// TIA Portal V17 export
// export: Created 2022-07-20T07:02:31.4890995Z, ExportSetting WithDefaults, DisplayName Totally Integrated Automation Portal, DisplayVersion V17, DisplayName TIA Portal Openness, DisplayVersion V17, DisplayName TIA Portal Version Control Interface, DisplayVersion V17, DisplayName SINAMICS Startdrive Advanced, DisplayVersion V17, DisplayName SINAMICS Startdrive G130, G150, S120, S150, SINAMICS MV, S210, DisplayVersion V17, DisplayName SINAMICS Startdrive G110M, G120, G120C, G120D, G120P, G115D, DisplayVersion V17, DisplayName STEP 7 Professional, DisplayVersion V17, DisplayName STEP 7 Safety, DisplayVersion V17, DisplayName WinCC Advanced, DisplayVersion V17
FUNCTION_BLOCK "FB11004_ProfileDataFifo"   // FB11004, LAD
TITLE = FIFO
{ S7_Optimized_Access := 'TRUE' }
VERSION : 0.1
// stored: AutoNumber false, IsIECCheckEnabled false, IsRetainMemResEnabled false, MemoryReserve 100, SetENOAutomatically false, UDAEnableTagReadback false
   VAR_INPUT
      GetProfile { ExternalAccessible := 'False'; ExternalVisible := 'False'; ExternalWritable := 'False'} : Bool;
      State { ExternalAccessible := 'False'; ExternalVisible := 'False'; ExternalWritable := 'False'} : UInt;
      Profile { ExternalAccessible := 'False'; ExternalVisible := 'False'; ExternalWritable := 'False'} : "stSheetProfile";
   END_VAR
   VAR_OUTPUT
      ItemsNumber { ExternalAccessible := 'False'; ExternalVisible := 'False'; ExternalWritable := 'False'} : UInt;
      ProfileAvailable { ExternalAccessible := 'False'; ExternalVisible := 'False'; ExternalWritable := 'False'} : Bool;
      Status { ExternalAccessible := 'False'; ExternalVisible := 'False'; ExternalWritable := 'False'} : UInt;
      ActualProfile { ExternalAccessible := 'False'; ExternalVisible := 'False'; ExternalWritable := 'False'} : "stSheetProfile";
   END_VAR
   VAR
      statFifo : Array[1.."MAX_IFOIL_FIFO_ITEMS_NUMBER"] of "stSheetProfile";
      statItemNumber { S7_SetPoint := 'True'} : UInt := 0;
      R_TRIG_GetProfile : R_TRIG;
      R_TRIG_GetDataFifo { S7_SetPoint := 'True'} : R_TRIG;
      statLastItem { S7_SetPoint := 'True'} : Bool;
   END_VAR
   VAR_TEMP
      FifoNumber : UInt;   // NextProfileTo
      AreaNumber : UInt;
   END_VAR
BEGIN

REGION Network 1 (SCL): Comments
   //==========================================================================================
   // SIEMENS SAS      RC-FR DI FA APC
   //------------------------------------------------------------------------------------------
   // Restrictions:    TIA V16 and more
   // Requirements:    S7-1500 - MGI Library
   // Functionality:   This function block offers fifo functionnality for stSheetProfile
   //------------------------------------------------------------------------------------------
   // Change log table:
   // Version      Date        Expert in charge    Changes applied
   // 01.00.01     09.06.2020  RTO                 First released version
   //==========================================================================================
END_REGION

REGION Network 2 (SCL): First Scan
   IF "FirstScan" THEN

       // Clear Interface
       #Status := 16#0;
       #ItemsNumber := "MAX_IFOIL_FIFO_ITEMS_NUMBER";
       #ProfileAvailable := FALSE;

       #ActualProfile.Length := 0.0;
       #ActualProfile.StampAreaStartAdjustment := 0.0;
       FOR #AreaNumber := 1 TO "MAX_NUMBER_OF_FOIL_AREA" DO
           #ActualProfile.Area[#AreaNumber].Start := 0.0;
           #ActualProfile.Area[#AreaNumber].End := 0.0;
       END_FOR;

       // Clear Fifo
       FOR #FifoNumber := 1 TO "MAX_IFOIL_FIFO_ITEMS_NUMBER" DO
           #statFifo[#FifoNumber].Length := 0.0;
           #statFifo[#FifoNumber].StampAreaStartAdjustment := 0.0;
           FOR #AreaNumber := 1 TO "MAX_NUMBER_OF_FOIL_AREA" DO
               #statFifo[#FifoNumber].Area[#AreaNumber].Start := 0.0;
               #statFifo[#FifoNumber].Area[#AreaNumber].End := 0.0;
           END_FOR;
       END_FOR;

       #statItemNumber := 0;
       #statLastItem := FALSE;

   END_IF;
END_REGION

REGION Network 3 (SCL): Edge Signal Management
   REGION EDGE SIGNALS
       #R_TRIG_GetProfile(CLK := #GetProfile);
       #R_TRIG_GetDataFifo(CLK := #State = 1 AND #statItemNumber < "MAX_IFOIL_FIFO_ITEMS_NUMBER" AND NOT #R_TRIG_GetProfile.Q);
   END_REGION
END_REGION

REGION Network 4 (SCL): Manage Fifo ready
   IF #State = 0 AND (#Status = 1 OR #Status = 2)
   THEN
       #Status := 0;
   END_IF;
END_REGION

REGION Network 5 (SCL): Put data in Fifo
   IF #State = 1 AND #statItemNumber < "MAX_IFOIL_FIFO_ITEMS_NUMBER" AND NOT #R_TRIG_GetProfile.Q THEN

       IF #R_TRIG_GetDataFifo.Q THEN
           // Get profile
           #statFifo[#statItemNumber + 1] := #Profile;

           // increase number of items
           #statItemNumber := #statItemNumber + 1;

       END_IF;

       // Send status
       #Status := 1;
   END_IF;
END_REGION

REGION Network 6 (SCL): Clear Fifo data
   IF #State = 2 AND #statItemNumber > 0 AND NOT #R_TRIG_GetProfile.Q THEN

       // Clear Fifo
       FOR #FifoNumber := 1 TO "MAX_IFOIL_FIFO_ITEMS_NUMBER" DO
           #statFifo[#FifoNumber].Length := 0.0;
           #statFifo[#FifoNumber].StampAreaStartAdjustment := 0.0;
           FOR #AreaNumber := 1 TO "MAX_NUMBER_OF_FOIL_AREA" DO
               #statFifo[#FifoNumber].Area[#AreaNumber].Start := 0.0;
               #statFifo[#FifoNumber].Area[#AreaNumber].End := 0.0;
           END_FOR;
       END_FOR;

       // Reset number of items
       #statItemNumber := 0;

       // Send status
       #Status := 2;

   END_IF;
END_REGION

REGION Network 7 (SCL): Get data from Fifo
   IF #R_TRIG_GetProfile.Q THEN

       // Get profile in Fifo
       #ActualProfile := #statFifo[1];

       IF #statItemNumber >= 2 THEN
           // Go up values in Fifo
           FOR #FifoNumber := 2 TO #statItemNumber DO
               #statFifo[#FifoNumber - 1] := #statFifo[#FifoNumber];
           END_FOR;
       END_IF;

       // Check if last item
       #statLastItem := #statItemNumber = 1;

       IF #statItemNumber >= 1 THEN
           // Clear last profile
           #statFifo[#statItemNumber].Length := 0.0;
           #statFifo[#statItemNumber].StampAreaStartAdjustment := 0.0;
           FOR #AreaNumber := 1 TO "MAX_NUMBER_OF_FOIL_AREA" DO
               #statFifo[#statItemNumber].Area[#AreaNumber].Start := 0.0;
               #statFifo[#statItemNumber].Area[#AreaNumber].End := 0.0;
           END_FOR;

           // Decrease number of items
           #statItemNumber := #statItemNumber - 1;
       END_IF;

   END_IF;
END_REGION

REGION Network 8: Manage profile available information
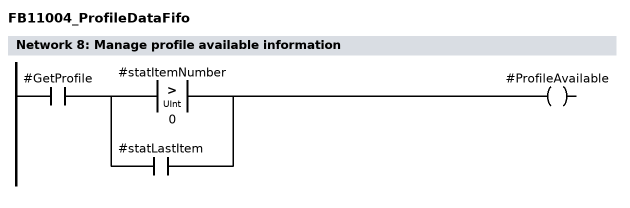
   RUNG wire#powerrail
      Contact( #GetProfile )
      wire#w1
      { S7_Templates := "SrcType := UInt" } GT_Contact(in1 := #statItemNumber, in2 := 0)
      wire#w2
      Coil( #ProfileAvailable )
   END_RUNG
   RUNG wire#w1
      Contact( #statLastItem )
   END_RUNG wire#w2
   // the same network as SCL:
   #ProfileAvailable := #GetProfile AND ((#statItemNumber > 0) OR #statLastItem);
END_REGION

REGION Network 9 (SCL): Manage number of items available
   #ItemsNumber := "MAX_IFOIL_FIFO_ITEMS_NUMBER" - #statItemNumber;
END_REGION
END_FUNCTION_BLOCK
